// SIMATIC STEP 7 (V5.x) project TEMA 13 EJRCICIO 32
// CPU: CPU313 C-2 DP(1)
// station: P_ADR_BUS
// station: Hardware
// station: Equipo SIMATIC 300
// program: Programa S7(1)

SYMBOL_TABLE
"FLANCOS"	DB 1	DB 1
"MANIOBRA"	DB 2	DB 2
"P DERECHA"	I 0.0	BOOL
"P IZQUIERDA"	I 0.1	BOOL
"P PARO"	I 0.2	BOOL
"TERMICO"	I 0.3	BOOL
"Cycle Execution"	OB 1	OB 1
"M DERECHA"	Q 0.0	BOOL
"LED DERECHA"	Q 0.1	BOOL
"M IZQUIERDA"	Q 0.2	BOOL
"LED IZQUIERDA"	Q 0.3	BOOL
"LED PARO"	Q 0.4	BOOL
"LED AVERIA"	Q 0.5	BOOL
END_SYMBOL_TABLE

DATA_BLOCK "FLANCOS"	// DB 1
VERSION : 0.1
  STRUCT
   M0 : BOOL ;
   M1 : BOOL ;
   M2 : BOOL ;
   M3 : BOOL ;
   M4 : BOOL ;
   M5 : BOOL ;
   M6 : BOOL ;
   M7 : BOOL ;
   M10 : BOOL ;
   M11 : BOOL ;
   M12 : BOOL ;
   M13 : BOOL ;
   M14 : BOOL ;
   M15 : BOOL ;
   M16 : BOOL ;
   M17 : BOOL ;
   M20 : BOOL ;
   M21 : BOOL ;
   M22 : BOOL ;
   M23 : BOOL ;
   M24 : BOOL ;
   M25 : BOOL ;
   M26 : BOOL ;
   M27 : BOOL ;
  END_STRUCT ;	
BEGIN
END_DATA_BLOCK

DATA_BLOCK "MANIOBRA"	// DB 2
VERSION : 0.1
  STRUCT
   MARCA0 : BOOL ;
   MARCA1 : BOOL ;
   MARCA2 : BOOL ;
   MARCA3 : BOOL ;
   MARCA4 : BOOL ;
   MARCA5 : BOOL ;
   MARCA6 : BOOL ;
   MARCA7 : BOOL ;
   MARCA10 : BOOL ;
   MARCA11 : BOOL ;
   MARCA12 : BOOL ;
   MARCA13 : BOOL ;
   MARCA14 : BOOL ;
  END_STRUCT ;	
BEGIN
END_DATA_BLOCK

ORGANIZATION_BLOCK "Cycle Execution"	// OB 1
TITLE = "Main Program Sweep (Cycle)"
//INVERSION DE GIRO TEMPORIZADA SIN PASAR POR PAR0 Y NORMAL PASANDO POR PARO
VERSION : 0.1
VAR_TEMP
  OB1_EV_CLASS : BYTE ;	//Bits 0-3 = 1 (Coming event), Bits 4-7 = 1 (Event class 1)
  OB1_SCAN_1 : BYTE ;	//1 (Cold restart scan 1 of OB 1), 3 (Scan 2-n of OB 1)
  OB1_PRIORITY : BYTE ;	//Priority of OB Execution
  OB1_OB_NUMBR : BYTE ;	//1 (Organization block 1, OB1)
  OB1_RESERVED_1 : BYTE ;	//Reserved for system
  OB1_RESERVED_2 : BYTE ;	//Reserved for system
  OB1_PREV_CYCLE : INT ;	//Cycle time of previous OB1 scan (milliseconds)
  OB1_MIN_CYCLE : INT ;	//Minimum cycle time of OB1 (milliseconds)
  OB1_MAX_CYCLE : INT ;	//Maximum cycle time of OB1 (milliseconds)
  OB1_DATE_TIME : DATE_AND_TIME ;	//Date and time OB1 started
END_VAR
BEGIN
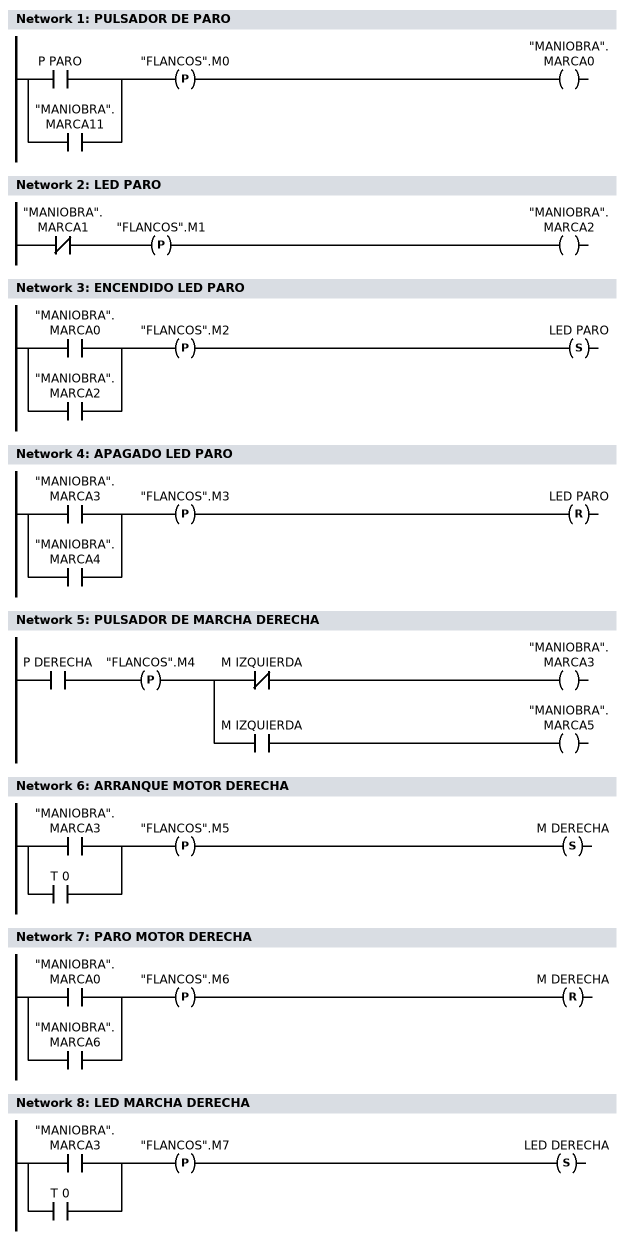
NETWORK
TITLE = PULSADOR DE PARO
      A(;
      O     "P PARO";
      O     "MANIOBRA".MARCA11;
      );
      FP    "FLANCOS".M0;
      =     "MANIOBRA".MARCA0;
NETWORK
TITLE = LED PARO
      AN    "MANIOBRA".MARCA1;
      FP    "FLANCOS".M1;
      =     "MANIOBRA".MARCA2;
NETWORK
TITLE = ENCENDIDO LED PARO
      A(;
      O     "MANIOBRA".MARCA0;
      O     "MANIOBRA".MARCA2;
      );
      FP    "FLANCOS".M2;
      S     "LED PARO";
NETWORK
TITLE = APAGADO LED PARO
      A(;
      O     "MANIOBRA".MARCA3;
      O     "MANIOBRA".MARCA4;
      );
      FP    "FLANCOS".M3;
      R     "LED PARO";
NETWORK
TITLE = PULSADOR DE MARCHA DERECHA
      A     "P DERECHA";
      FP    "FLANCOS".M4;
      =     L 20.0;
      A     L 20.0;
      AN    "M IZQUIERDA";
      =     "MANIOBRA".MARCA3;
      A     L 20.0;
      A     "M IZQUIERDA";
      =     "MANIOBRA".MARCA5;
NETWORK
TITLE = ARRANQUE MOTOR DERECHA
      A(;
      O     "MANIOBRA".MARCA3;
      O     T 0;
      );
      FP    "FLANCOS".M5;
      S     "M DERECHA";
NETWORK
TITLE = PARO MOTOR DERECHA
      A(;
      O     "MANIOBRA".MARCA0;
      O     "MANIOBRA".MARCA6;
      );
      FP    "FLANCOS".M6;
      R     "M DERECHA";
NETWORK
TITLE = LED MARCHA DERECHA
      A(;
      O     "MANIOBRA".MARCA3;
      O     T 0;
      );
      FP    "FLANCOS".M7;
      S     "LED DERECHA";
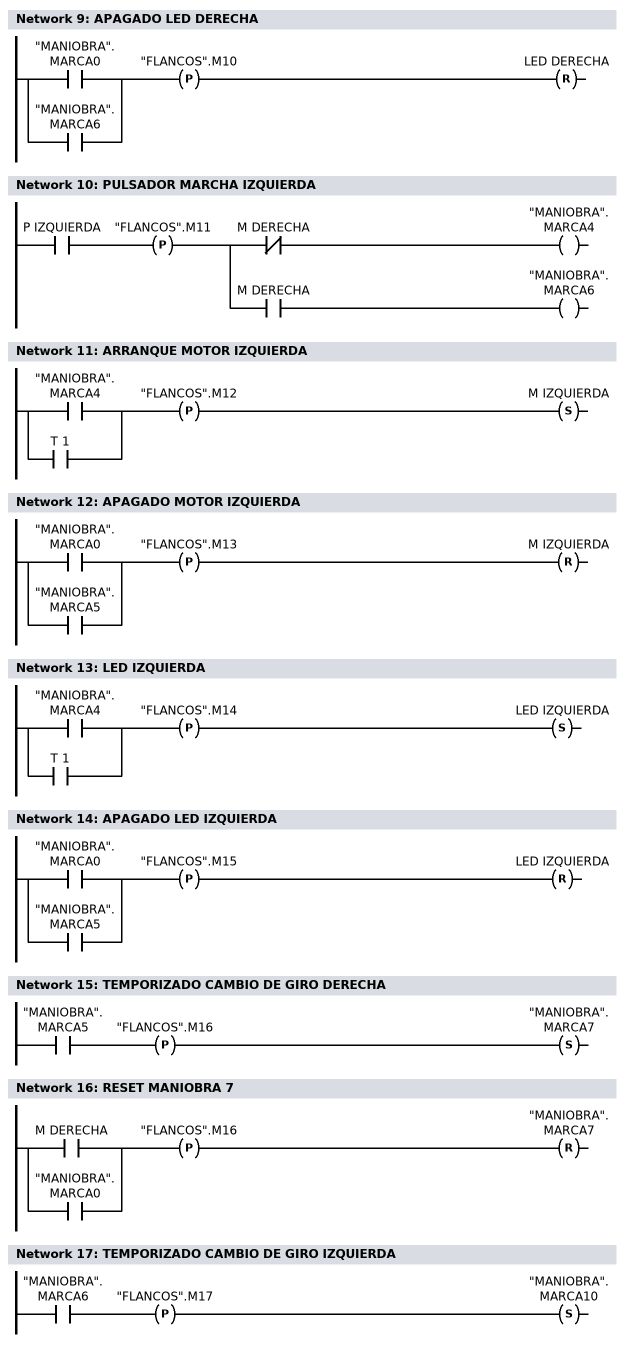
NETWORK
TITLE = APAGADO LED DERECHA 
      A(;
      O     "MANIOBRA".MARCA0;
      O     "MANIOBRA".MARCA6;
      );
      FP    "FLANCOS".M10;
      R     "LED DERECHA";
NETWORK
TITLE = PULSADOR MARCHA IZQUIERDA
      A     "P IZQUIERDA";
      FP    "FLANCOS".M11;
      =     L 20.0;
      A     L 20.0;
      AN    "M DERECHA";
      =     "MANIOBRA".MARCA4;
      A     L 20.0;
      A     "M DERECHA";
      =     "MANIOBRA".MARCA6;
NETWORK
TITLE = ARRANQUE MOTOR IZQUIERDA
      A(;
      O     "MANIOBRA".MARCA4;
      O     T 1;
      );
      FP    "FLANCOS".M12;
      S     "M IZQUIERDA";
NETWORK
TITLE = APAGADO MOTOR IZQUIERDA
      A(;
      O     "MANIOBRA".MARCA0;
      O     "MANIOBRA".MARCA5;
      );
      FP    "FLANCOS".M13;
      R     "M IZQUIERDA";
NETWORK
TITLE = LED IZQUIERDA
      A(;
      O     "MANIOBRA".MARCA4;
      O     T 1;
      );
      FP    "FLANCOS".M14;
      S     "LED IZQUIERDA";
NETWORK
TITLE = APAGADO LED IZQUIERDA
      A(;
      O     "MANIOBRA".MARCA0;
      O     "MANIOBRA".MARCA5;
      );
      FP    "FLANCOS".M15;
      R     "LED IZQUIERDA";
NETWORK
TITLE = TEMPORIZADO CAMBIO DE GIRO DERECHA
//DESCONECTA EL SENTIDO CONTRARIO Y AL CABO DE 3 SEG. CONECTA EL SENTIDO 
//ELEGIDO.ESTA MARCA DE MANIOBRA MANTIENE EL FLUJO DE CORRIENTE ININTERRUMPIDA 
//PARA QUE PUEDE ACTUAR EL T0
      A     "MANIOBRA".MARCA5;
      FP    "FLANCOS".M16;
      S     "MANIOBRA".MARCA7;
NETWORK
TITLE = RESET MANIOBRA 7
      A(;
      O     "M DERECHA";
      O     "MANIOBRA".MARCA0;
      );
      FP    "FLANCOS".M16;
      R     "MANIOBRA".MARCA7;
NETWORK
TITLE = TEMPORIZADO CAMBIO DE GIRO IZQUIERDA
//FUNCIONA DE LA MISMA FORMA QUE LA COMENTADA ANTERIORMENTE QUE T1
      A     "MANIOBRA".MARCA6;
      FP    "FLANCOS".M17;
      S     "MANIOBRA".MARCA10;
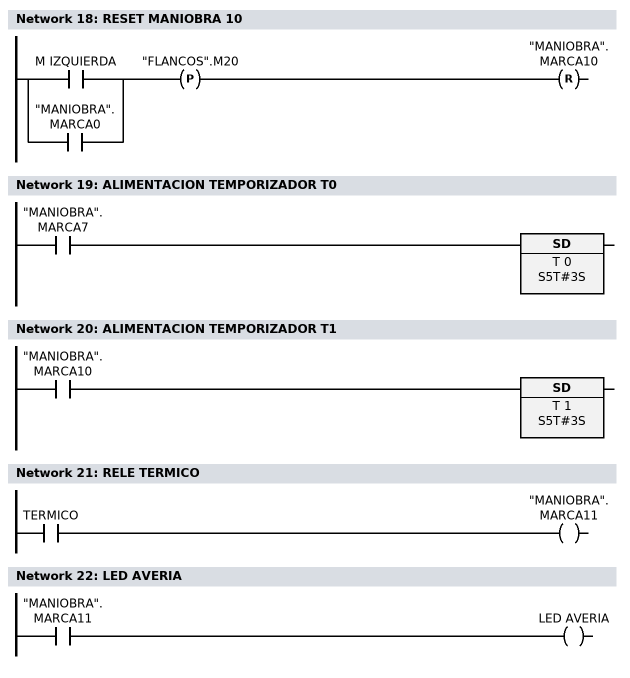
NETWORK
TITLE = RESET MANIOBRA 10
      A(;
      O     "M IZQUIERDA";
      O     "MANIOBRA".MARCA0;
      );
      FP    "FLANCOS".M20;
      R     "MANIOBRA".MARCA10;
NETWORK
TITLE = ALIMENTACION TEMPORIZADOR T0 
      A     "MANIOBRA".MARCA7;
      L     S5T#3S;
      SD    T 0;
NETWORK
TITLE = ALIMENTACION TEMPORIZADOR T1
      A     "MANIOBRA".MARCA10;
      L     S5T#3S;
      SD    T 1;
NETWORK
TITLE = RELE TERMICO
      A     "TERMICO";
      =     "MANIOBRA".MARCA11;
NETWORK
TITLE = LED AVERIA
      A     "MANIOBRA".MARCA11;
      =     "LED AVERIA";
END_ORGANIZATION_BLOCK
